PROGRAM selectPos020
VAR
END_VAR


gvl.cfgPos_OF020:= gvl_p.aPositionsE020[gvl.actPos].numOF;
gvl.cfgPos_LT020:= gvl_p.aPositionsE020[gvl.actPos].lote;
gvl.cfgPos_Class020:= gvl_p.aPositionsE020[gvl.actPos].class;
gvl.cfgPos_Pot020:= gvl_p.aPositionsE020[gvl.actPos].pot;
gvl.cfgPos_Reat020:= gvl_p.aPositionsE020[gvl.actPos].reator;

END_PROGRAM

(* stored: Version 1.1.0.1, ProductVersion 3.1.4024.12
   POU selectPos020: Id {037432fc-182e-4ae1-8ba6-b7c470ab61e0}, SpecialFunc None *)
